Staubli VAL3: MsgRecvState.dtx

public num RECEIVE_HEADER
public num DECODE_HEADER
public num RECEIVE_BODY
public num DECODE_BODY
public num PUSH_MOTION
public num HANDLE_REQUEST
public num SEND_ACK
